// TIA Portal V19 export
TYPE "LEXCHANGETRAY_typePlasticEm5_toRollerRecieve"
// stored: Access Published
   STRUCT
      feedback { S7_SetPoint := 'True'} : "LEXCHANGETRAY_typeRoller_toWorkStationRollerFeedback_B2";
      req { S7_SetPoint := 'True'} : "LEXCHANGETRAY_typeRoller_toWorkStationRollerReq_B2";
   END_STRUCT;
END_TYPE
